{attribute 'qualified_only'}
{attribute 'strict'}
///Cylinder enable mode
TYPE E_MotorEnableMode :
(
    eMotorEnaOff,       ///Enable does not affect motor
    eMotorEnaAll,       ///When enable false, motor cannot move CW or CCW
    eMotorEnaAllowCW,   ///When enable false, motor can onlu move CW
    eMotorEnaAllowCCW   ///When enable false, motor can onlu move CCW   
);
END_TYPE

(* stored: Version 1.1.0.1, ProductVersion 3.1.4019.2
   DUT E_MotorEnableMode: Id {15f5c0b2-ec4a-417f-b8f7-17df33db6769} *)
